TYPE ST_CamSeq :
STRUCT
	rAxisX			:REAL;
	rAxisY			:REAL;
	nCamProg		:UINT;
	bExecute		:BOOL;
END_STRUCT
END_TYPE

(* stored: Version 1.1.0.1, ProductVersion 3.1.4024.10
   DUT ST_CamSeq: Id {631dd778-95e1-44cf-989b-01ded73d051a} *)
